VAR_GLOBAL
	Clock 						: TClock;
	Config 						: TConfig;
	configuring					: BOOL;
	config_request				: BOOL;
	Config_Message				: STRING(300);
	config_speed				: INT:=1;
	List_of_Recipes				: ARRAY[1..10] OF Recipe;
END_VAR

(* stored: Version 1.1.0.1, ProductVersion 3.1.4020.12
   GVL GVL_Objects: Id {065d5605-db40-49f0-8c53-de89a8f7f7d0} *)
